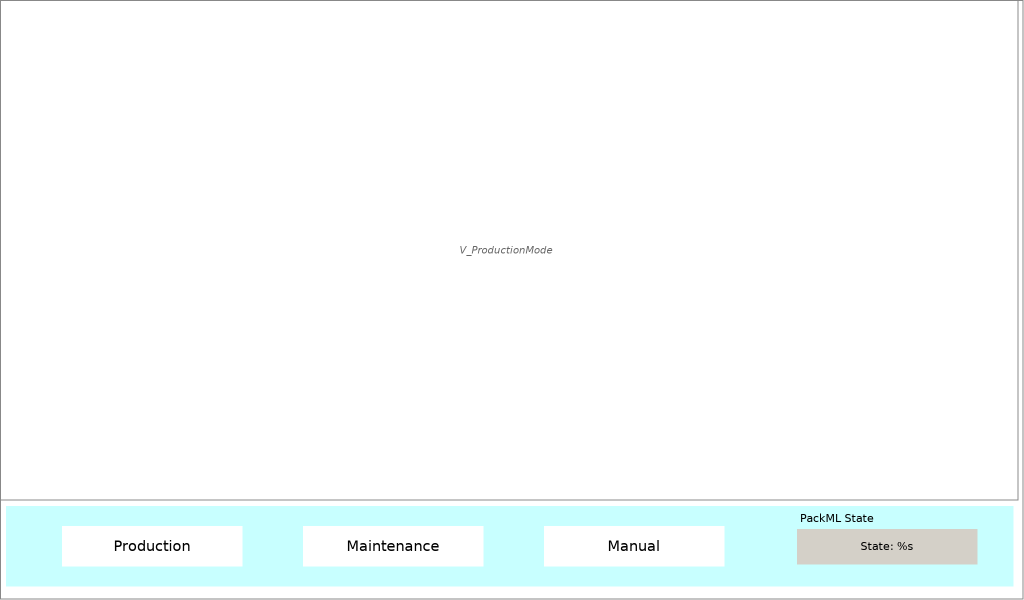
VISUALIZATION V_MainMenu  // 1024x600
VAR_IN_OUT
	HMI : ST_PackMLBaseModule_HMI;
	HMIAxeX : ST_AxisBase_HMI;
	HMI_Recipe : ST_RecipeBuilder_HMI;
	HMI2 : ST_Machine_HMI;
END_VAR
    RoundedRectangle (5,505 1009x82)
    Textfield (797,529 180x35), "State: %s", text variable: HMI2.Status.PackMLState
    RoundedRectangle (62,526 180x40), "Production", colour toggle: HMI.Status.Mode = E_PMLUnitMode.ePMLUnitMode_Production
        OnMouseClick: execute { HMI.Command.Mode := E_PMLUnitMode.ePMLUnitMode_Production; }
    RoundedRectangle (303,526 180x40), "Maintenance", colour toggle: HMI.Status.Mode = E_PMLUnitMode.ePMLUnitMode_Maintenance
        OnMouseClick: execute { HMI.Command.Mode := E_PMLUnitMode.ePMLUnitMode_Maintenance; }
    RoundedRectangle (544,526 180x40), "Manual", colour toggle: HMI.Status.Mode = E_PMLUnitMode.ePMLUnitMode_Manual
        OnMouseClick: execute { HMI.Command.Mode := E_PMLUnitMode.ePMLUnitMode_Manual; }
    Frame (-6,0 1024x500), frame switch variable: GVL_HMI.MenuToDisplay
        shows V_ProductionMode(HMI := MAIN.Seedra.PackMLBaseModule_HMI, HMI_GantryXYZ := MAIN.Seedra.GantryXYZ.GantryXYZ_HMI, HMI_Recipe := MAIN.Seedra.RecipeConfig_HMI)
        shows V_ManualMode(HMI := MAIN.Seedra.PackMLBaseModule_HMI, HMIAxeX := MAIN.Seedra.GantryXYZ.AxisX.AxisBase_HMI, HMIAxeY := MAIN.Seedra.GantryXYZ.AxisY.AxisBase_HMI, HMIAxeZ := MAIN.Seedra.GantryXYZ.AxisZ.AxisBase_HMI)
        shows V_MaintenanceMode(HMI := MAIN.Seedra.PackMLBaseModule_HMI, HMI_GantryXYZ := MAIN.Seedra.GantryXYZ.GantryXYZ_HMI)
    Label (788,498 98x41), "PackML State"
END_VISUALIZATION

(* stored: Version 1.1.0.1, ProductVersion 3.1.4024.15
   Visu V_MainMenu: Id {a579ab76-3dfa-0e50-1e72-1a62fe47c520} *)
